FUNCTION_BLOCK AUI_SEL_AX (* Adapter Selection: Plug OUT = (G.D1 ? IN1 : IN0) *)
  (* Standard: 61499-2; Description: Copyright (c) 2026 HR Agrartechnik GmbH This program and the accompanying materials are made available under the terms of the Eclipse Public License 2.0 which is available at https://www.eclipse.org/legal/epl-2.0/ SPDX-License-Identifier: EPL-2.0 *)
  (* Version 1.0, 2026-04-19, Franz Höpfinger, HR Agrartechnik GmbH, initial API and implementation *)
  PACKAGE adapter::iec61131::selection;
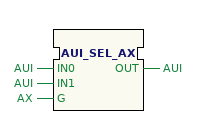
  SOCKETS
    IN0 : adapter::types::unidirectional::AUI; (* Input 0 (selected if G is FALSE) *)
    IN1 : adapter::types::unidirectional::AUI; (* Input 1 (selected if G is TRUE) *)
    G : adapter::types::unidirectional::AX; (* Selector *)
  END_SOCKETS
  PLUGS
    OUT : adapter::types::unidirectional::AUI; (* Selected Output *)
  END_PLUGS
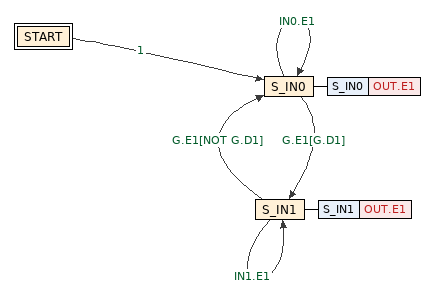
  EC_STATES
    START; (* Initial State *)
    S_IN0 : S_IN0 -> OUT.E1; (* Process Selection *)
    S_IN1 : S_IN1 -> OUT.E1;
  END_STATES
  EC_TRANSITIONS
    START TO S_IN0 := 1;
    S_IN1 TO S_IN0 := G.E1[NOT G.D1];
    S_IN0 TO S_IN1 := G.E1[G.D1];
    S_IN0 TO S_IN0 := IN0.E1;
    S_IN1 TO S_IN1 := IN1.E1;
  END_TRANSITIONS
  ALGORITHM S_IN0 IN ST: (* dd *)
OUT.D1 := IN0.D1;
  END_ALGORITHM
  ALGORITHM S_IN1 IN ST: (* dd *)
OUT.D1 := IN1.D1;
  END_ALGORITHM
END_FUNCTION_BLOCK
